FUNCTION_BLOCK NetLinkParametersFB
VAR_INPUT
END_VAR
VAR_OUTPUT
END_VAR
VAR
END_VAR

METHOD Update : BOOL
VAR_INPUT
	Parameters: REFERENCE TO GreenMasterBaseParameters;
END_VAR
END_METHOD

END_FUNCTION_BLOCK

(* stored: Version 1.1.0.1, ProductVersion 3.1.4024.6
   POU NetLinkParametersFB: Id {70d71791-c95b-4941-80ac-0ecb7778050c}, SpecialFunc None
   Method Update: Id {d2b89ff4-bc7c-4576-a53f-0863be15f6a0} *)
